PROGRAM P_NormalizeJointVel
VAR
	fbActuatorVelToNormalized4 : FB_ActuatorVelFeedForward;
END_VAR


// Going from joint velocity to normalized signal inn PID
fbActuatorVelToNormalized4(fActuatorVelocity := G_InverseKinematics.fq4Dotref,
							fMaxActuatorVelocity := 0.030, //m/s
							fVelocityFeedForward => G_Servo.fNormalizedActuatorVelFeedForward_q4Dot);

END_PROGRAM

(* stored: Version 1.1.0.1, ProductVersion 3.1.4024.12
   POU P_NormalizeJointVel: Id {9d2f287e-2610-4fe5-b68c-866cfdd65833}, SpecialFunc None *)
